Fanuc KAREL source: kt00068.KL

-- PROVISIONAL review KL for V940-1; original PC SHA256 b44711800ceeb7adadd80712cce993054cfe0184837eec7081a2f692525ce368
-- Incomplete behavior may be omitted. Consult companion uncertainty JSON. Do not deploy.
PROGRAM KT00068
%NOLOCKGROUP
VAR
  I1 : INTEGER
  R2 : REAL
  OUT : REAL
BEGIN
  -- V9_ZERO_TABLE_METADATA_HINT layout=0001; no indexed target words; source/name/runtime held
  -- UNRESOLVED_PC offsets 5-16; opcodes 2E,23
  -- UNRESOLVED_PC offsets 21-32; opcodes 2E,23
  -- UNRESOLVED_PC offsets 37-58; opcodes 21,21,29,64,6B,23
  -- UNRESOLVED_PC offsets 63-67; opcodes 7F
END KT00068
